{attribute 'GeneratedUsingTerminal: EL3681-0000-0017'}
{attribute addProperty BoxType "EL3681-0000-0017"}
{attribute addProperty Id "SettingAT %I*Setting_24C049402"}
{attribute addProperty CRC "3273657976"}
{attribute addProperty Size "2"}
TYPE SAI_Range_C3200E78 EXTENDS InputBase_8311D824 :
STRUCT
	{attribute addProperty Name "Setting"}
	Setting AT %I* : Setting_24C04940;
END_STRUCT
END_TYPE

(* stored: Version 1.2.0.0, ProductVersion 3.1.4024.9
   DUT SAI_Range_C3200E78: Id {4cb08ccf-e95b-4993-9f5b-461703eedec7} *)
